// TwinCAT 3 PLC project Untitled1
// ProgramVersion: 3.1.4023.0
// libraries:
//   Tc2_Standard, * (Beckhoff Automation GmbH)
//   Tc2_System, * (Beckhoff Automation GmbH)
//   Tc3_Module, * (Beckhoff Automation GmbH)
// project tree:
//   DUTs/ Axis.TcDUT, Robot.TcDUT
//   GVLs/ GVL.TcGVL
//   / PlcTask.TcTTO
//   POUs/ MAIN.TcPOU
// real-time tasks:
//   TASK PlcTask: cycle T#10ms, priority 20, ADS port 350

CONFIGURATION Untitled1
    RESOURCE PLC ON TwinCAT3
        TASK PlcTask(INTERVAL := T#10ms, PRIORITY := 20);
        PROGRAM MAIN WITH PlcTask : MAIN;
    END_RESOURCE
END_CONFIGURATION

// ---- DUTs/Axis.TcDUT
TYPE Axis :
STRUCT
	
	X: REAL;
	Y: REAL;
	Z: REAL;
	
END_STRUCT
END_TYPE

// ---- DUTs/Robot.TcDUT
TYPE Robot :
STRUCT
	Manual_Mode_Enabled: BOOL;
		
	Rotor_Axis: Axis; 
	Finger_Axis: Axis;
	Wrist_Axis: Axis;
	Forearm_Axis: Axis; 
	PistonIK_Axis: Axis;
	Piston_Axis: Axis;
	Arm_Axis: Axis;
	CylinderIK_Axis: Axis;
	Cylinder_Axis: Axis; 

END_STRUCT
END_TYPE

// ---- GVLs/GVL.TcGVL
{attribute 'qualified_only'}
VAR_GLOBAL

	Test_Axis: Axis; 
	
	RobotVars : Robot;
	
END_VAR

// ---- POUs/MAIN.TcPOU
PROGRAM MAIN
VAR
END_VAR

END_PROGRAM
